{attribute 'GeneratedUsingTerminal: CU1123-0010-0016'}
{attribute addProperty BoxType "CU1123-0010-0016"}
{attribute addProperty Id "A_0003_CU1124_0000_0016A_0003_CU1124_0000_0016_D1C35140124"}
{attribute addProperty CRC "1415063249"}
{attribute addProperty Size "124"}
TYPE A_0002_CU1123_0010_0016_545826D1 EXTENDS CU1123_AB5A9467 :
STRUCT
	{attribute addProperty Name "A_0003_CU1124_0000_0016"}
	{attribute addProperty PreviousPort "A_0002(CU1123-0010-0016) : D"}
	A_0003_CU1124_0000_0016 : A_0003_CU1124_0000_0016_D1C35140;
END_STRUCT
END_TYPE

(* stored: Version 1.2.0.0, ProductVersion 3.1.4024.9
   DUT A_0002_CU1123_0010_0016_545826D1: Id {03738218-d4c0-402f-b3b4-3316275d9a42} *)
